{attribute addProperty BoxType "EK1100-0000-0018"}
{attribute addProperty Id "TcTerminals210_2BK1250TcTerminals210_2BK1250_0898888900"}
{attribute addProperty CRC "3182404534"}
{attribute addProperty SizeInBites "0"}
{attribute addProperty SizeInBytes "0"}
TYPE TcTerminals210_2EK1100_BDAFA3B6 EXTENDS EK1100_179A0949 :
STRUCT
	{attribute addProperty Name "TcTerminals210_2BK1250"}
	TcTerminals210_2BK1250 : TcTerminals210_2BK1250_08988889;
END_STRUCT
END_TYPE

(* stored: Version 1.2.0.0, ProductVersion 3.1.4024.9
   DUT TcTerminals210_2EK1100_BDAFA3B6: Id {35341998-f9b4-4d11-bc86-fb3e5a367990} *)
